{attribute 'GeneratedUsingTerminal: EL5032-0000-0021'}
{attribute addProperty BoxType "EL5032-0000-0021"}
{attribute addProperty Id "EtcSlaveTerminalBaseFB_Inputs_Channel_1AT %I*FB_Inputs_Channel_7405098814FB_Inputs_Channel_2AT %I*FB_Inputs_Channel_7405098814WcStateAT %I*WcState_9091E0EB2InfoDataAT %I*InfoData_32EB74EA10"}
{attribute addProperty CRC "2028036765"}
{attribute addProperty Size "40"}
TYPE EL5032_78E1629D EXTENDS EtcSlaveTerminalBase :
STRUCT
	{attribute addProperty Name "FB_Inputs_Channel_1"}
	FB_Inputs_Channel_1 : FB_Inputs_Channel_74050988;
	{attribute addProperty Name "FB_Inputs_Channel_2"}
	FB_Inputs_Channel_2 : FB_Inputs_Channel_74050988;
	{attribute addProperty Name "WcState"}
	WcState : WcState_9091E0EB;
	{attribute addProperty Name "InfoData"}
	InfoData : InfoData_32EB74EA;
END_STRUCT
END_TYPE

(* stored: Version 1.2.0.0, ProductVersion 3.1.4024.9
   DUT EL5032_78E1629D: Id {c7c29c25-3216-4fbf-bc62-11dc917fc291} *)
